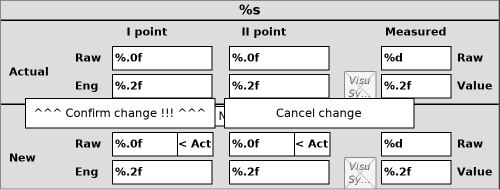
VISUALIZATION MeasureCalibration  // 500x190
VAR_IN_OUT
	stMeasureData:stMeasurementScalingData;
END_VAR
VAR_INPUT
	diAnalogIn:DINT;
	MeasureName:STRING;
END_VAR
VAR
	rRaw1:REAL;
	rRaw2:REAL:= 32767;
	rEng1:REAL;
	rEng2:REAL;
	bConfirmation:BOOL:=FALSE;
END_VAR
    Rectangle (0,20 500x84)
    Rectangle (112,46 100x24), "%.0f", text variable: stMeasureData.rScalingRawValue_I, input disabled if: TRUE
    Label (72,46 40x24), "Raw"
    Rectangle (112,74 100x24), "%.2f", text variable: stMeasureData.rScalingEngValue_I, input disabled if: TRUE
    Label (72,74 40x24), "Eng"
    Label (112,20 70x24), "I point"
    Rectangle (229,46 100x24), "%.0f", text variable: stMeasureData.rScalingRawValue_II, input disabled if: TRUE
    Rectangle (229,74 100x24), "%.2f", text variable: stMeasureData.rScalingEngValue_II, input disabled if: TRUE
    Label (229,20 70x24), "II point"
    Image (344,71 32x32), image: VisuSymbols.Symbols.ArrowBoldRight
    Label (381,20 70x24), "Measured"
    Rectangle (381,74 70x24), "%.2f", text variable: ( (DINT_TO_REAL(diAnalogIn) - stMeasureData.rScalingRawValue_I)/ ( LIMIT(0.1,(stMeasureData.rScalingRawValue_II - stMeasureData.rScalingRawValue_I),999999999999)))*( stMeasureData.rScalingEngValue_II - stMeasureData.rScalingEngValue_I)+stMeasureData.rScalingEngValue_I, input disabled if: TRUE
    Rectangle (381,46 70x24), "%d", text variable: diAnalogIn, input disabled if: TRUE
    Label (454,46 40x24), "Raw"
    Label (454,74 40x24), "Value"
    Rectangle (0,104 500x85)
    Rectangle (112,132 68x24), "%.0f", text variable: rRaw1
        OnMouseClick: write rRaw1 via Default, title 'New Raw I value', format %.0f
    Label (72,132 40x24), "Raw"
    Rectangle (112,160 100x24), "%.2f", text variable: rEng1
        OnMouseClick: write rEng1 via Default, title 'New Eng I value', format %.2f
    Label (72,160 40x24), "Eng"
    Rectangle (229,132 68x24), "%.0f", text variable: rRaw2
        OnMouseClick: write rRaw2 via Default, title 'New Raw II value', format %.0f
    Rectangle (229,160 100x24), "%.2f", text variable: rEng2
        OnMouseClick: write rEng2 via Default, title 'New Eng II value', format %.2f
    Image (344,157 32x32), image: VisuSymbols.Symbols.ArrowBoldRight
    Rectangle (381,160 70x24), "%.2f", text variable: ( (DINT_TO_REAL(diAnalogIn) - rRaw1)/ (LIMIT(1,(rRaw2 - rRaw1),9999999999999) ) ) * ( rEng2 - rEng1)+ rEng1, input disabled if: TRUE
    Rectangle (381,132 70x24), "%d", text variable: diAnalogIn, input disabled if: TRUE
    Label (454,132 40x24), "Raw"
    Label (454,160 40x24), "Value"
    Label (6,146 40x24), "New"
    Label (6,60 40x24), "Actual"
    RoundedRectangle (113,106 216x20), "^^ Set NEW ^^", invisible if: bConfirmation
        toggle bConfirmation
    RoundedRectangle (177,132 36x24), "< Act"
        OnMouseClick: execute { rRaw1:= DINT_TO_REAL(diAnalogIn); }
    RoundedRectangle (294,132 36x24), "< Act"
        OnMouseClick: execute { rRaw2 := DINT_TO_REAL(diAnalogIn); }
    RoundedRectangle (25,98 190x30), "^^^ Confirm change !!! ^^^", invisible if: NOT bConfirmation
        OnMouseClick: execute {
            stMeasureData.rScalingEngValue_I := rEng1;
            stMeasureData.rScalingEngValue_II := rEng2;
            stMeasureData.rScalingRawValue_I := rRaw1;
            stMeasureData.rScalingRawValue_II := rRaw2;
            bConfirmation:= FALSE;
        }
    RoundedRectangle (224,98 190x30), "Cancel change", invisible if: NOT bConfirmation
        OnMouseClick: execute { bConfirmation:= FALSE; }
    Rectangle (0,0 500x20), "%s", text variable: MeasureName
END_VISUALIZATION

(* stored: Version 1.1.0.1, ProductVersion 3.1.4024.12
   Visu MeasureCalibration: Id {184c0f3c-927f-4f61-8e68-249e4d31b497} *)
